{attribute 'GeneratedUsingTerminal: AX8206-0100-0101-0101'}
{attribute addProperty BoxType "AX8206-0100-0101-0101"}
{attribute addProperty Id "EtcSlaveTerminalBaseDeviceDevice_6E2575772Device_SafetyDevice_Safety_C21945A160Ch_ACh_A_1FF86D8522Ch_BCh_B_5E084BAA22WcStateAT %I*WcState_B516A2644InfoDataAT %I*InfoData_386C00A526"}
{attribute addProperty CRC "1825383343"}
{attribute addProperty Size "136"}
TYPE AX8206_6CCD23AF EXTENDS EtcSlaveTerminalBase :
STRUCT
	{attribute addProperty Name "Device"}
	Device : Device_6E257577;
	{attribute addProperty Name "Device_Safety"}
	Device_Safety : Device_Safety_C21945A1;
	{attribute addProperty Name "Ch_A"}
	Ch_A : Ch_A_1FF86D85;
	{attribute addProperty Name "Ch_B"}
	Ch_B : Ch_B_5E084BAA;
	{attribute addProperty Name "WcState"}
	WcState : WcState_B516A264;
	{attribute addProperty Name "InfoData"}
	InfoData : InfoData_386C00A5;
END_STRUCT
END_TYPE

(* stored: Version 1.2.0.0, ProductVersion 3.1.4024.9
   DUT AX8206_6CCD23AF: Id {cf1298af-4cf5-4e77-8237-bd8e3ef72fe7} *)
